FUNCTION_BLOCK StandardRoom EXTENDS BaseRoom
VAR_INPUT
	rTemperature	: LREAL := 20.0 + Math.Random();
END_VAR
VAR    	
    // Entity
    _entityExtend	: EntityExtend(_entityStart);
	
    _lowTemperature : Room_State_LowTemperature(_ctx, rTemperature);
    _demand         : Room_State_DemandHeating(_ctx);
   
    _entityEnd2		: EntityEnd;
END_VAR

METHOD Execute
SUPER^.Execute();

// Simulation
IF NOT sim.bTick THEN
	RETURN;
END_IF

IF bInletValve AND bOutletValve THEN
	rTemperature := rTemperature + sim.param.rRoomTemperatureRisePerHeater * Math.Random();
END_IF

rTemperature := rTemperature + sim.param.rRoomTemperaturePassiveDrop * Math.Random();

IF rTemperature < 0 THEN
	rTemperature := 0;
ELSIF rTemperature > 100 THEN
	rTemperature := 100;
END_IF
END_METHOD

END_FUNCTION_BLOCK

(* stored: Version 1.1.0.1
   POU StandardRoom: Id {2e0e75c6-de15-4761-ae40-14041f36bdf4}, SpecialFunc None
   Method Execute: Id {51b956d4-c76f-41de-a458-174fed593c72} *)
